// TIA Portal V17 export
// export: Created 2025-08-05T09:35:58.4846759Z, ExportSetting WithDefaults, DisplayName Totally Integrated Automation Portal, DisplayVersion V17, DisplayName TIA Portal Openness, DisplayVersion V17, DisplayName TIA Portal Version Control Interface, DisplayVersion V17, DisplayName SINAMICS Startdrive Advanced, DisplayVersion V17, DisplayName SINAMICS Startdrive G130, G150, S120, S150, SINAMICS MV, S210, DisplayVersion V17, DisplayName SINAMICS Startdrive G110M, G120, G120C, G120D, G120P, G115D, DisplayVersion V17, DisplayName STEP 7 Professional, DisplayVersion V17, DisplayName STEP 7 Safety, DisplayVersion V17, DisplayName WinCC Advanced, DisplayVersion V17
DATA_BLOCK "FgLaser1Control"   // DB180
TITLE = FG $[name] Control system / FG $[name] Steuerung
{ S7_Optimized_Access := 'TRUE'; DB_Accessible_From_OPC_UA := 'FALSE' }
FAMILY : FG
VERSION : 0.0.0.0
// FG $[name] Control system / FG $[name] Steuerung
// stored: AutoNumber true, DBAccessibleFromOPCUA false, DBAccessibleFromWebserver true, IsOnlyStoredInLoadMemory false, IsRetainMemResEnabled false, IsWriteProtectedInAS false, MemoryReserve 100
   VAR
      general { ExternalAccessible := 'False'; ExternalVisible := 'False'; ExternalWritable := 'False'} : "typeFgControlGeneral";   // FG Laser 1: Allgemein / FG Laser 1: general
      activeJob { ExternalAccessible := 'False'; ExternalVisible := 'False'; ExternalWritable := 'False'} : Struct   // FG Laser 1: Aktiver Auftrag / FG Laser 1: active job
         job1SealAirOn { ExternalAccessible := 'False'; ExternalVisible := 'False'; ExternalWritable := 'False'} : Bool;   // FG Laser 1 - Auftrag 1: Sperrluft einschalten aktiv / FG Laser 1 - job 1: switch on sealing air active
         job2LaserOn { ExternalAccessible := 'False'; ExternalVisible := 'False'; ExternalWritable := 'False'} : Bool;   // FG Laser 1 - Auftrag 2: Laser ein aktiv / FG Laser 1 - job 2: laser on active
         job3SealAirOff { ExternalAccessible := 'False'; ExternalVisible := 'False'; ExternalWritable := 'False'} : Bool;   // FG Laser 1 - Auftrag 3: Sperrluft ausschalten aktiv / FG Laser 1 - job 3: switch off sealing air active
         job4LaserOnSpecialFunction { ExternalAccessible := 'False'; ExternalVisible := 'False'; ExternalWritable := 'False'} : Bool;   // FG Laser 1 - Auftrag 4: Laser ein Sonderablauf aktiv / FG Laser 1 - job 4: laser on special sequence active
         job99ToHomePos { ExternalAccessible := 'False'; ExternalVisible := 'False'; ExternalWritable := 'False'} : Bool;   // FG Laser 1 - Auftrag 99: Zur Grundstellung aktiv / FG Laser 1 - Job 99: To home position active
      END_STRUCT;
      motions { ExternalAccessible := 'False'; ExternalVisible := 'False'; ExternalWritable := 'False'} : Struct   // FG Laser 1: Bewegungen / FG laser 1: Motions
         switchOnSealAir { ExternalAccessible := 'False'; ExternalVisible := 'False'; ExternalWritable := 'False'} : "typeMotion";   // FG Laser 1: Sperrluft einschalten / FG Laser 1: Switch on sealing air
         switchOffSealAir { ExternalAccessible := 'False'; ExternalVisible := 'False'; ExternalWritable := 'False'} : "typeMotion";   // FG Laser 1: Sperrluft ausschalten / FG Laser 1: Switch off sealing air
         switchOnProtectionGas1_1 { ExternalAccessible := 'False'; ExternalVisible := 'False'; ExternalWritable := 'False'} : "typeMotion";   // FG Laser 1: Schutzgas 1.1 einschalten / FG laser 1: Switch on shielding gas 1.1
         switchOffProtectionGas1_1 { ExternalAccessible := 'False'; ExternalVisible := 'False'; ExternalWritable := 'False'} : "typeMotion";   // FG Laser 1: Schutzgas 1.1 ausschalten / FG laser 1: Switch off shielding gas 1.1
         switchOnProtectionGas1_2 { ExternalAccessible := 'False'; ExternalVisible := 'False'; ExternalWritable := 'False'} : "typeMotion";   // FG Laser 1: Schutzgas 1.2 einschalten / FG laser 1: Switch on shielding gas 1.2
         switchOffProtectionGas1_2 { ExternalAccessible := 'False'; ExternalVisible := 'False'; ExternalWritable := 'False'} : "typeMotion";   // FG Laser 1: Schutzgas 1.2 ausschalten / FG laser 1: Switch off shielding gas 1.2
         switchOnProtectionGas1_3 { ExternalAccessible := 'False'; ExternalVisible := 'False'; ExternalWritable := 'False'} : "typeMotion";   // FG Laser 1: Schutzgas 1.3 einschalten / FG laser 1: Switch on shielding gas 1.3
         switchOffProtectionGas1_3 { ExternalAccessible := 'False'; ExternalVisible := 'False'; ExternalWritable := 'False'} : "typeMotion";   // FG Laser 1: Schutzgas 1.3 ausschalten / FG laser 1: Switch off shielding gas 1.3
         switchOnProtectionGas1_4 { ExternalAccessible := 'False'; ExternalVisible := 'False'; ExternalWritable := 'False'} : "typeMotion";   // FG Laser 1: Schutzgas 1.4 einschalten / FG laser 1: Switch on shielding gas 1.4
         switchOffProtectionGas1_4 { ExternalAccessible := 'False'; ExternalVisible := 'False'; ExternalWritable := 'False'} : "typeMotion";   // FG Laser 1: Schutzgas 1.4 ausschalten / FG laser 1: Switch off shielding gas 1.4
         switchOnProtectionGas1_5 { ExternalAccessible := 'False'; ExternalVisible := 'False'; ExternalWritable := 'False'} : "typeMotion";   // FG Laser 1: Schutzgas 1.5 einschalten / FG laser 1: Switch on shielding gas 1.5
         switchOffProtectionGas1_5 { ExternalAccessible := 'False'; ExternalVisible := 'False'; ExternalWritable := 'False'} : "typeMotion";   // FG Laser 1: Schutzgas 1.5 ausschalten / FG laser 1: Switch off shielding gas 1.5
         switchOnProtectionGas1_6 { ExternalAccessible := 'False'; ExternalVisible := 'False'; ExternalWritable := 'False'} : "typeMotion";   // FG Laser 1: Schutzgas 1.6 einschalten / FG laser 1: Switch on shielding gas 1.6
         switchOffProtectionGas1_6 { ExternalAccessible := 'False'; ExternalVisible := 'False'; ExternalWritable := 'False'} : "typeMotion";   // FG Laser 1: Schutzgas 1.6 ausschalten / FG laser 1: Switch off shielding gas 1.6
         switchOnProtectionGasCalibration { ExternalAccessible := 'False'; ExternalVisible := 'False'; ExternalWritable := 'False'} : "typeMotion";   // FG Laser 1: Schutzgas Kalibriersystem einschalten / FG laser 1: Switch on shielding gas calibration system
         switchOffProtectionGasComplete { ExternalAccessible := 'False'; ExternalVisible := 'False'; ExternalWritable := 'False'} : "typeMotion";   // FG Laser 1: Schutzgas Laser 1 komplett ausschalten
         switchOffProtectionGasCalibration { ExternalAccessible := 'False'; ExternalVisible := 'False'; ExternalWritable := 'False'} : "typeMotion";   // FG Laser 1: Schutzgas Kalibriersystem ausschalten / FG laser 1: Switch off shielding gas calibration system
      END_STRUCT;
      laserTaskCurrent { ExternalAccessible := 'False'; ExternalVisible := 'False'; ExternalWritable := 'False'} : Bool;   // FG Laser 1: Laser Task Aktiv / FG Laser 1: Laser task active
      laserEvaluationNotActive { ExternalAccessible := 'False'; ExternalVisible := 'False'; ExternalWritable := 'False'} : Bool;   // FG Laser 1: Laser Auswertung nicht aktiv / FG Laser 1: Laser evaluation not active
   END_VAR
   VAR RETAIN
      laserMeasuring { ExternalAccessible := 'False'; ExternalVisible := 'False'; ExternalWritable := 'False'} : Struct   // FG Laser 1: Lasermessungen / FG laser 1: Laser measurements
         powerMeasuringRequest { ExternalAccessible := 'False'; ExternalVisible := 'False'; ExternalWritable := 'False'} : Bool;   // FG Laser 1: Laserleistungsmessung Anforderung / FG laser 1: laser power measurement request
         powerMeasuringStart { ExternalAccessible := 'False'; ExternalVisible := 'False'; ExternalWritable := 'False'} : Bool;   // FG Laser 1: Laserleistungsmessung starten / FG laser 1: Start laser power measurement
         powerMeasuringDone { ExternalAccessible := 'False'; ExternalVisible := 'False'; ExternalWritable := 'False'} : Bool;   // FG Laser 1: Laserleistungsmessung beendet / FG laser 1: laser power measurement not completed
         beamWatchMeasuringRequest { ExternalAccessible := 'False'; ExternalVisible := 'False'; ExternalWritable := 'False'} : Bool;   // FG Laser 1: BeamWatchmessung Anforderung / FG laser 1: BeamWatchmeasurement request
         beamWatchMeasuringStart { ExternalAccessible := 'False'; ExternalVisible := 'False'; ExternalWritable := 'False'} : Bool;   // FG Laser 1: BeamWatchmessung starten / FG Laser 1: Start Beamwatch measurement
         beamWatchMeasuringDone { ExternalAccessible := 'False'; ExternalVisible := 'False'; ExternalWritable := 'False'} : Bool;   // FG Laser 1: BeamWatchmessung beendet / FG laser 1: BeamWatchmeasurement not finished
         lddCalibrationRequest { ExternalAccessible := 'False'; ExternalVisible := 'False'; ExternalWritable := 'False'} : Bool;   // FG Laser 1: LDD Kalibrierung Anforderung / FG laser 1: LDD calibration request
         lddCalibrationStart { ExternalAccessible := 'False'; ExternalVisible := 'False'; ExternalWritable := 'False'} : Bool;   // FG Laser 1: LDD Kalibrierung starten / FG laser 1: start LDD calibration
         lddCalibrationDone { ExternalAccessible := 'False'; ExternalVisible := 'False'; ExternalWritable := 'False'} : Bool;   // FG Laser 1: LDD Kalibrierung beendet / FG laser 1: LDD calibration not finished
         changeCalibrationPieceDone { ExternalAccessible := 'False'; ExternalVisible := 'False'; ExternalWritable := 'False'} : Bool;   // FG Laser 1: Opferblech LDD Kalibrierung tauschen beendet / FG laser 1: Change sacrificial part LDD calibration finished
         ready { ExternalAccessible := 'False'; ExternalVisible := 'False'; ExternalWritable := 'False'} : Bool;   // FG Laser 1: Lasermessung bereit / FG laser 1: Laser measurement ready
      END_STRUCT;
   END_VAR
   VAR
      dryRunWeldSimDone { ExternalAccessible := 'False'; ExternalVisible := 'False'; ExternalWritable := 'False'} : Bool;   // FG Laser 1: Trockenlauf der Schweißsimulation durchgeführt / FG laser 1: dry run of welding simulation performed
      dryRunWeldSimOk { ExternalAccessible := 'False'; ExternalVisible := 'False'; ExternalWritable := 'False'} : Bool := TRUE;   // FG Laser 1: Ergebnis der Trockenschweißung: Aufgabe einstellen OK / FG laser 1: result of dry welding: set task OK
      SMCstatus { ExternalAccessible := 'False'; ExternalVisible := 'False'; ExternalWritable := 'False'} : "typeSmcChillerHrle90a40cmStatus";   // FG Laser 1: SMC Kühler / FG Laser 1: SMC cooler
      laserManOnBypassEnable { ExternalAccessible := 'False'; ExternalVisible := 'False'; ExternalWritable := 'False'} : Bool;   // FG Laser 1: Aktiviert die Umgehung einiger Regeln, um den Laser einzuschalten / FG Laser 1: Activates the bypass of some rules to switch on the laser
   END_VAR
   VAR RETAIN
      analogSensor { ExternalAccessible := 'False'; ExternalVisible := 'False'; ExternalWritable := 'False'} : Struct   // FG Laser 1: Analogsensoren
         FlowProtGas1_1 { ExternalAccessible := 'False'; ExternalVisible := 'False'; ExternalWritable := 'False'} : Struct   // FG Laser 1: Durchflusssensor Schutzgas 1.1
            limitsSensor { ExternalAccessible := 'False'; ExternalVisible := 'False'; ExternalWritable := 'False'} : "typeAnalogSensorUniversalLimits";   // FG Laser 1: Durchflusssensor Schutzgas 1.1 Limits
            positionsSensor { ExternalAccessible := 'False'; ExternalVisible := 'False'; ExternalWritable := 'False'} : "typeAnalogSensorUniversalPositions";   // FG Laser 1: Durchflusssensor Schutzgas 1.1 Positionen
         END_STRUCT;
         FlowProtGas1_2 { ExternalAccessible := 'False'; ExternalVisible := 'False'; ExternalWritable := 'False'} : Struct   // FG Laser 1: Durchflusssensor Schutzgas 1.2
            limitsSensor { ExternalAccessible := 'False'; ExternalVisible := 'False'; ExternalWritable := 'False'} : "typeAnalogSensorUniversalLimits";   // FG Laser 1: Durchflusssensor Schutzgas 1.2 Limits
            positionsSensor { ExternalAccessible := 'False'; ExternalVisible := 'False'; ExternalWritable := 'False'} : "typeAnalogSensorUniversalPositions";   // FG Laser 1: Durchflusssensor Schutzgas 1.2 Positionen
         END_STRUCT;
         FlowProtGas1_3 { ExternalAccessible := 'False'; ExternalVisible := 'False'; ExternalWritable := 'False'} : Struct   // FG Laser 1: Durchflusssensor Schutzgas 1.3
            limitsSensor { ExternalAccessible := 'False'; ExternalVisible := 'False'; ExternalWritable := 'False'} : "typeAnalogSensorUniversalLimits";   // FG Laser 1: Durchflusssensor Schutzgas 1.3 Limits
            positionsSensor { ExternalAccessible := 'False'; ExternalVisible := 'False'; ExternalWritable := 'False'} : "typeAnalogSensorUniversalPositions";   // FG Laser 1: Durchflusssensor Schutzgas 1.3 Positionen
         END_STRUCT;
         FlowProtGas1_4 { ExternalAccessible := 'False'; ExternalVisible := 'False'; ExternalWritable := 'False'} : Struct   // FG Laser 1: Durchflusssensor Schutzgas 1.4
            limitsSensor { ExternalAccessible := 'False'; ExternalVisible := 'False'; ExternalWritable := 'False'} : "typeAnalogSensorUniversalLimits";   // FG Laser 1: Durchflusssensor Schutzgas 1.4 Limits
            positionsSensor { ExternalAccessible := 'False'; ExternalVisible := 'False'; ExternalWritable := 'False'} : "typeAnalogSensorUniversalPositions";   // FG Laser 1: Durchflusssensor Schutzgas 1.4 Positionen
         END_STRUCT;
         FlowProtGas1_5 { ExternalAccessible := 'False'; ExternalVisible := 'False'; ExternalWritable := 'False'} : Struct   // FG Laser 1: Durchflusssensor Schutzgas 1.5
            limitsSensor { ExternalAccessible := 'False'; ExternalVisible := 'False'; ExternalWritable := 'False'} : "typeAnalogSensorUniversalLimits";   // FG Laser 1: Durchflusssensor Schutzgas 1.5 Limits
            positionsSensor { ExternalAccessible := 'False'; ExternalVisible := 'False'; ExternalWritable := 'False'} : "typeAnalogSensorUniversalPositions";   // FG Laser 1: Durchflusssensor Schutzgas 1.5 Positionen
         END_STRUCT;
         FlowProtGas1_6 { ExternalAccessible := 'False'; ExternalVisible := 'False'; ExternalWritable := 'False'} : Struct   // FG Laser 1: Durchflusssensor Schutzgas 1.6
            limitsSensor { ExternalAccessible := 'False'; ExternalVisible := 'False'; ExternalWritable := 'False'} : "typeAnalogSensorUniversalLimits";   // FG Laser 1: Durchflusssensor Schutzgas 1.6 Limits
            positionsSensor { ExternalAccessible := 'False'; ExternalVisible := 'False'; ExternalWritable := 'False'} : "typeAnalogSensorUniversalPositions";   // FG Laser 1: Durchflusssensor Schutzgas 1.6 Positionen
         END_STRUCT;
      END_STRUCT;
   END_VAR
   VAR
      UsageCounterCalibrationPiece { ExternalAccessible := 'False'; ExternalVisible := 'False'; ExternalWritable := 'False'} : Struct   // FG Laser 1: Verschleisszähler Opferblech 1 / FG laser 1: wear counter sacrificial plate 1
         prewarning { ExternalAccessible := 'False'; ExternalVisible := 'False'; ExternalWritable := 'False'} : Bool;   // FG Laser 1: Vorwarnung des Zählers für Opferblech 1 / FG laser 1: prewarning of counter for sacrificial plate 1
         warning { ExternalAccessible := 'False'; ExternalVisible := 'False'; ExternalWritable := 'False'} : Bool;   // FG Laser 1: Warnung des Zählers für Opferblech 1 / FG laser 1: warning of counter for sacrificial plate 1
         error { ExternalAccessible := 'False'; ExternalVisible := 'False'; ExternalWritable := 'False'} : Bool;   // FG Laser 1: Zähler für Opferblech 1 erreicht / FG laser 1: counter for sacrificial plate 1 reached
      END_STRUCT;
      UsageCounterProtectionGlass { ExternalAccessible := 'False'; ExternalVisible := 'False'; ExternalWritable := 'False'} : Struct   // FG Laser 1: Verschleißzähler Schutglas / FG laser 1: wear counter protective glass
         prewarning { ExternalAccessible := 'False'; ExternalVisible := 'False'; ExternalWritable := 'False'} : Bool;   // FG Laser 1: Vorwarnung des Zählers für Schutzglas Laser 1 / FG laser 1: prewarning of counter for protective glass laser 1
         warning { ExternalAccessible := 'False'; ExternalVisible := 'False'; ExternalWritable := 'False'} : Bool;   // FG Laser 1: Warnung des Zählers für Schutglas Laser 1 / FG laser 1: warning of counter for protective glass laser 1
         error { ExternalAccessible := 'False'; ExternalVisible := 'False'; ExternalWritable := 'False'} : Bool;   // FG Laser 1: Zähler für Schutzglas erreicht Laser 1 / FG laser 1: counter for protective glass reached laser 1
      END_STRUCT;
      CalibrationPieceChanged { ExternalAccessible := 'False'; ExternalVisible := 'False'; ExternalWritable := 'False'} : Bool;   // FG Laser 1: Opferblech muss getauscht werden / FG laser 1: sacrificial plate must be replaced
   END_VAR
BEGIN
   // motions.switchOnSealAir.inPosition : FG Laser 1: Sperrluft eingeschalten / FG Laser 1: Sealing air switched on
   // motions.switchOnSealAir.autoInPos : FG Laser 1: Sperrluft eingeschalten (Automatic) / FG Laser 1: Sealing air switched on (automatic)
   // motions.switchOffSealAir.inPosition : FG Laser 1: Sperrluft ausgeschalten / FG Laser 1: Sealing air switched off
   // motions.switchOffSealAir.autoInPos : FG Laser 1: Sperrluft ausgeschalten (Automatic) / FG Laser 1: Sealing air switched off (automatic)
   // motions.switchOnProtectionGas1_1.inPosition : FG Laser 1: Schutzgas 1.1 eingeschalten / FG laser 1: Shielding gas 1.1 switched on
   // motions.switchOnProtectionGas1_1.autoInPos : FG Laser 1: Schutzgas 1.1 eingeschalten (Automatic) / FG laser 1: Shielding gas 1.1 switched on (automatic)
   // motions.switchOffProtectionGas1_1.inPosition : FG Laser 1: Schutzgas 1.1 ausgeschalten / FG laser 1: Shielding gas 1.1 switched off
   // motions.switchOffProtectionGas1_1.autoInPos : FG Laser 1: Schutzgas 1.1 ausgeschalten (Automatic) / FG laser 1: Shielding gas 1.1 switched off (automatic)
   // motions.switchOnProtectionGas1_2.inPosition : FG Laser 1: Schutzgas 1.2 eingeschalten / FG laser 1: Shielding gas 1.2 switched on
   // motions.switchOnProtectionGas1_2.autoInPos : FG Laser 1: Schutzgas 1.2 eingeschalten (Automatic) / FG laser 1: Shielding gas 1.2 switched on (automatic)
   // motions.switchOffProtectionGas1_2.inPosition : FG Laser 1: Schutzgas 1.2 ausgeschalten / FG laser 1: Shielding gas 1.2 switched off
   // motions.switchOffProtectionGas1_2.autoInPos : FG Laser 1: Schutzgas 1.2 ausgeschalten (Automatic) / FG laser 1: Shielding gas 1.2 switched off (automatic)
   // motions.switchOnProtectionGas1_3.inPosition : FG Laser 1: Schutzgas 1.3 eingeschalten / FG laser 1: Shielding gas 1.3 switched on
   // motions.switchOnProtectionGas1_3.autoInPos : FG Laser 1: Schutzgas 1.3 eingeschalten (Automatic) / FG laser 1: Shielding gas 1.3 switched on (automatic)
   // motions.switchOffProtectionGas1_3.inPosition : FG Laser 1: Schutzgas 1.3 ausgeschalten / FG laser 1: Shielding gas 1.3 switched off
   // motions.switchOffProtectionGas1_3.autoInPos : FG Laser 1: Schutzgas 1.3 ausgeschalten (Automatic) / FG laser 1: Shielding gas 1.3 switched off (automatic)
   // motions.switchOnProtectionGas1_4.inPosition : FG Laser 1: Schutzgas 1.4 eingeschalten / FG laser 1: Shielding gas 1.4 switched on
   // motions.switchOnProtectionGas1_4.autoInPos : FG Laser 1: Schutzgas 1.4 eingeschalten (Automatic) / FG laser 1: Shielding gas 1.4 switched on (automatic)
   // motions.switchOffProtectionGas1_4.inPosition : FG Laser 1: Schutzgas 1.4 ausgeschalten / FG laser 1: Shielding gas 1.4 switched off
   // motions.switchOffProtectionGas1_4.autoInPos : FG Laser 1: Schutzgas 1.4 ausgeschalten (Automatic) / FG laser 1: Shielding gas 1.4 switched off (automatic)
   // motions.switchOnProtectionGas1_5.inPosition : FG Laser 1: Schutzgas 1.5 eingeschalten / FG laser 1: Shielding gas 1.5 switched on
   // motions.switchOnProtectionGas1_5.autoInPos : FG Laser 1: Schutzgas 1.5 eingeschalten (Automatic) / FG laser 1: Shielding gas 1.5 switched on (automatic)
   // motions.switchOffProtectionGas1_5.inPosition : FG Laser 1: Schutzgas 1.5 ausgeschalten / FG laser 1: Shielding gas 1.5 switched off
   // motions.switchOffProtectionGas1_5.autoInPos : FG Laser 1: Schutzgas 1.5 ausgeschalten (Automatic) / FG laser 1: Shielding gas 1.5 switched off (automatic)
   // motions.switchOnProtectionGas1_6.inPosition : FG Laser 1: Schutzgas 1.6 eingeschalten / FG laser 1: Shielding gas 1.6 switched on
   // motions.switchOnProtectionGas1_6.autoInPos : FG Laser 1: Schutzgas 1.6 eingeschalten (Automatic) / FG laser 1: Shielding gas 1.6 switched on (automatic)
   // motions.switchOffProtectionGas1_6.inPosition : FG Laser 1: Schutzgas 1.6 ausgeschalten / FG laser 1: Shielding gas 1.6 switched off
   // motions.switchOffProtectionGas1_6.autoInPos : FG Laser 1: Schutzgas 1.6 ausgeschalten (Automatic) / FG laser 1: Shielding gas 1.6 switched off (automatic)
   // motions.switchOnProtectionGasCalibration.inPosition : FG Laser 1: Schutzgas Kalibriersystem eingeschalten / FG laser 1: Shielding gas calibration system switched on
   // motions.switchOnProtectionGasCalibration.autoInPos : FG Laser 1: Schutzgas Kalibriersystem eingeschalten (Automatic) / FG laser 1: Shielding gas calibration system switched on (automatic)
   // motions.switchOffProtectionGasComplete.inPosition : FG Laser 1: Schutzgas Kalibriersystem ausgeschalten / FG laser 1: Shielding gas calibration system switched off
   // motions.switchOffProtectionGasComplete.autoInPos : FG Laser 1: Schutzgas Kalibriersystem ausgeschalten (Automatic) / FG laser 1: Shielding gas calibration system switched off (automatic)
   // motions.switchOffProtectionGasCalibration.inPosition : FG Laser 1: Schutzgas Kalibriersystem ausgeschalten / FG laser 1: Shielding gas calibration system switched off
   // motions.switchOffProtectionGasCalibration.autoInPos : FG Laser 1: Schutzgas Kalibriersystem ausgeschalten (Automatic) / FG laser 1: Shielding gas calibration system switched off (automatic)
END_DATA_BLOCK
